{attribute 'GeneratedUsingTerminal: KL2531'}
{attribute addProperty BoxType "KL2531"}
{attribute addProperty Description ""}
{attribute addProperty Physics ""}
{attribute addProperty Id "Channel_1AT %Q*Channel_FEA3DBF80"}
{attribute addProperty CRC "3584972036"}
{attribute addProperty Size "0"}
TYPE KL2531_D5AE5504 :
STRUCT
	{attribute addProperty Name "Channel_1"}
	Channel_1 : Channel_FEA3DBF8;
END_STRUCT
END_TYPE

(* stored: Version 1.2.0.0, ProductVersion 3.1.4024.9
   DUT KL2531_D5AE5504: Id {9889742f-16b9-466c-9990-2c70e3fbb437} *)
